// TwinCAT 3 PLC project Controller
// ProgramVersion: 3.1.4026.25
// libraries:
//   Tc2_Standard, * (Beckhoff Automation GmbH)
//   Tc2_System, * (Beckhoff Automation GmbH)
// project tree:
//   / PlcTask.TcTTO
//   POUs/ MAIN.TcPOU
// real-time tasks:
//   TASK ModelTask: cycle T#10ms, priority 1, ADS port 350
//   TASK PlcTask: cycle T#1ms, priority 20, ADS port 351
// variable links:
//   Controller/Controller Instance <-> TcCOM Objects/SimIoMaster/SimIoGroup
//     PlcTask Inputs/MAIN.dx <-> Inputs/dx
//     PlcTask Inputs/MAIN.p <-> Inputs/p
//     PlcTask Inputs/MAIN.x <-> Inputs/x
//     PlcTask Outputs/MAIN.q <-> Outputs/q

CONFIGURATION Controller
    RESOURCE PLC ON TwinCAT3
        TASK PlcTask(INTERVAL := T#10ms, PRIORITY := 20);
        PROGRAM MAIN WITH PlcTask : MAIN;
    END_RESOURCE
END_CONFIGURATION

// ---- POUs/MAIN.TcPOU
PROGRAM MAIN
VAR
	// Controller inputs (system states)
	x  AT%I*  : LREAL := 0.0;	// State 1, Cylinder position	[m]
	dx AT%I*  : LREAL := 0.0;	// State 2, Cylinder velocity	[m s^-1]
	p  AT%I*  : LREAL := 0.0;	// State 3, Cylinder pressure	[Pa]

	// Controller outputs
	q  AT%Q*  : LREAL := 0.0;	// Input air flow				[m^3 s^-1]


	// Reference input
	w  : LREAL := 0.0;			// Cylinder position			[m]


	// Control canonical system states
	z1 : LREAL := 0.0;
	z2 : LREAL := 0.0;
	z3 : LREAL := 0.0;

	// Virtual controller output
	v  : LREAL := 0.0;


	// Piston parameter
	A  : LREAL := 5.0e-3;		// Piston area					[m^2]
	c  : LREAL := 2.0e3;		// Spring stiffness				[N m^-1]
	m  : LREAL := 1.0;			// Piston mass					[kg]

	// Controller design parameter
	L  : LREAL := -10.0;		// Desired closed loop eigenvalues
	r1 : LREAL := -L*L*L;		// Controller feedback gain 1
	r2 : LREAL := 3*L*L;		// Controller feedback gain 2
	r3 : LREAL := -3*L;			// Controller feedback gain 3
	f  : LREAL := -L*L*L;		// Controller input gain
END_VAR

// Control canonical system states
z1 := x;
z2 := dx;
z3 := -(c/m) * x + (A/m) * p;

// Virtual controller output
v := -r1 * z1 - r2 * z2 - r3 * z3 + f * w;

// Controller output
q := m * (x/p) * ((c/m)*dx + (A/m)*(dx*p/x) + v);

END_PROGRAM
